// TIA Portal V20 export
// export: Created 2026-07-16T23:20:30.0572279Z, ExportSetting WithDefaults, DisplayName Totally Integrated Automation Portal, DisplayVersion V20 Update 5, DisplayName TIA Portal Openness, DisplayVersion V20 Update 4, DisplayName TIA Portal Version Control Interface, DisplayVersion V20 Update 5, DisplayName SINAMICS Startdrive Advanced, DisplayVersion V20, DisplayName SINAMICS DCC, DisplayVersion V20, DisplayName SINAMICS Startdrive G130, G150, S120, S150, SINAMICS MV, G220, S200, S210, DisplayVersion V20, DisplayName SINAMICS Startdrive G110M, G120, G120C, G120D, G120P, G115D, DisplayVersion V20, DisplayName STEP 7 Professional, DisplayVersion V20 Update 5, DisplayName STEP 7 Safety, DisplayVersion V20 Update 2, DisplayName WinCC Basic/Comfort/Advanced, DisplayVersion V20 Update 5, DisplayName WinCC Unified, DisplayVersion V20 Update 5
FUNCTION "FC_ControlMain" : Void   // FC3, LAD
TITLE = Control Main
{ S7_Optimized_Access := 'TRUE' }
VERSION : 0.1
// Control area-Main (C-109): every cross-instance fact in the project lives here (C-127) - buffer-to-instance input wiring, the sequencer/motor/pusher calls in dependency order (sequencer decides, motor and pusher obey within the same scan), inter-instance command wiring, and the buffer output map. No working logic beyond wiring, with two documented extras (C-606): the In_Cycle lamp OR (owner ruling 2026-07-16, REQ-069 - field feedbacks, not commands) and the soft-start fault-reset pass-through to DQ11 (panel provides the output; Q-14 records the open control-on question).
// stored: AutoNumber true, IsIECCheckEnabled false, SetENOAutomatically false, UDAEnableTagReadback false
BEGIN

REGION Network 1: Sequencer Input Wiring
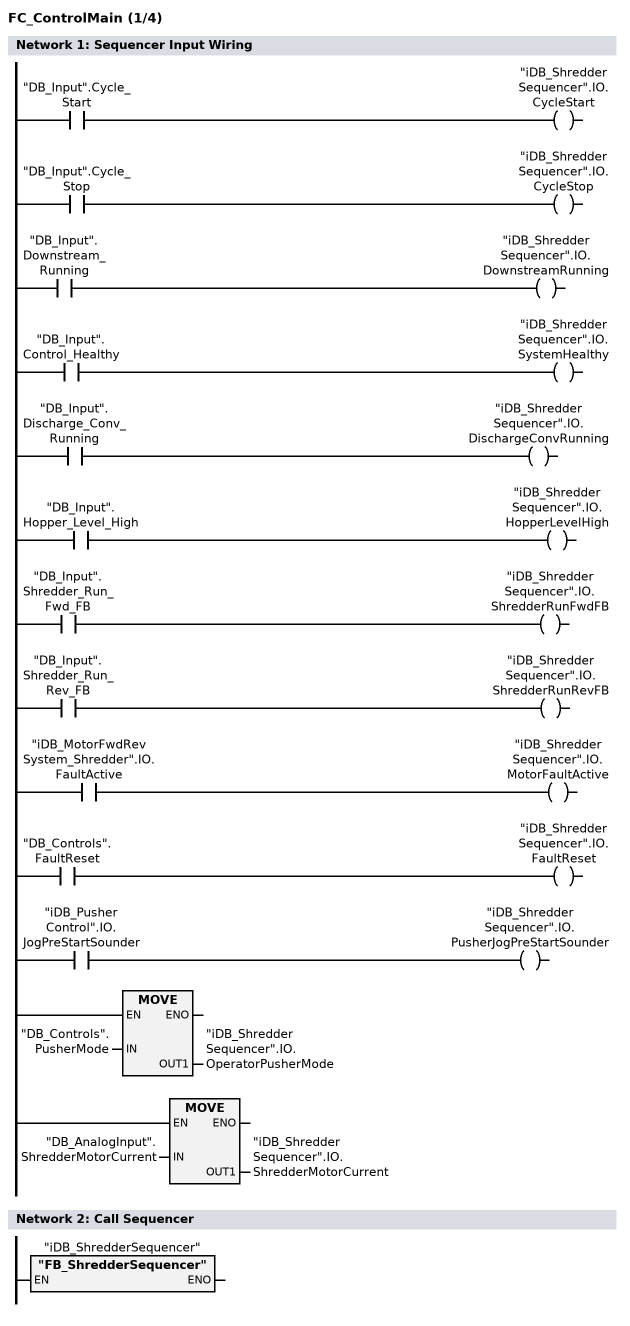
   RUNG wire#powerrail
      Contact( "DB_Input".Cycle_Start )
      Coil( "iDB_ShredderSequencer".IO.CycleStart )
   END_RUNG
   RUNG wire#powerrail
      Contact( "DB_Input".Cycle_Stop )
      Coil( "iDB_ShredderSequencer".IO.CycleStop )
   END_RUNG
   RUNG wire#powerrail
      Contact( "DB_Input".Downstream_Running )
      Coil( "iDB_ShredderSequencer".IO.DownstreamRunning )
   END_RUNG
   RUNG wire#powerrail
      Contact( "DB_Input".Control_Healthy )
      Coil( "iDB_ShredderSequencer".IO.SystemHealthy )
   END_RUNG
   RUNG wire#powerrail
      Contact( "DB_Input".Discharge_Conv_Running )
      Coil( "iDB_ShredderSequencer".IO.DischargeConvRunning )
   END_RUNG
   RUNG wire#powerrail
      Contact( "DB_Input".Hopper_Level_High )
      Coil( "iDB_ShredderSequencer".IO.HopperLevelHigh )
   END_RUNG
   RUNG wire#powerrail
      Contact( "DB_Input".Shredder_Run_Fwd_FB )
      Coil( "iDB_ShredderSequencer".IO.ShredderRunFwdFB )
   END_RUNG
   RUNG wire#powerrail
      Contact( "DB_Input".Shredder_Run_Rev_FB )
      Coil( "iDB_ShredderSequencer".IO.ShredderRunRevFB )
   END_RUNG
   RUNG wire#powerrail
      Contact( "iDB_MotorFwdRevSystem_Shredder".IO.FaultActive )
      Coil( "iDB_ShredderSequencer".IO.MotorFaultActive )
   END_RUNG
   RUNG wire#powerrail
      Contact( "DB_Controls".FaultReset )
      Coil( "iDB_ShredderSequencer".IO.FaultReset )
   END_RUNG
   RUNG wire#powerrail
      Contact( "iDB_PusherControl".IO.JogPreStartSounder )
      Coil( "iDB_ShredderSequencer".IO.PusherJogPreStartSounder )
   END_RUNG
   RUNG wire#powerrail
      Move(in := "DB_Controls".PusherMode, out1 => "iDB_ShredderSequencer".IO.OperatorPusherMode)
   END_RUNG
   RUNG wire#powerrail
      Move(in := "DB_AnalogInput".ShredderMotorCurrent, out1 => "iDB_ShredderSequencer".IO.ShredderMotorCurrent)
   END_RUNG
   // the same network as SCL:
   "iDB_ShredderSequencer".IO.CycleStart := "DB_Input".Cycle_Start;
   "iDB_ShredderSequencer".IO.CycleStop := "DB_Input".Cycle_Stop;
   "iDB_ShredderSequencer".IO.DownstreamRunning := "DB_Input".Downstream_Running;
   "iDB_ShredderSequencer".IO.SystemHealthy := "DB_Input".Control_Healthy;
   "iDB_ShredderSequencer".IO.DischargeConvRunning := "DB_Input".Discharge_Conv_Running;
   "iDB_ShredderSequencer".IO.HopperLevelHigh := "DB_Input".Hopper_Level_High;
   "iDB_ShredderSequencer".IO.ShredderRunFwdFB := "DB_Input".Shredder_Run_Fwd_FB;
   "iDB_ShredderSequencer".IO.ShredderRunRevFB := "DB_Input".Shredder_Run_Rev_FB;
   "iDB_ShredderSequencer".IO.MotorFaultActive := "iDB_MotorFwdRevSystem_Shredder".IO.FaultActive;
   "iDB_ShredderSequencer".IO.FaultReset := "DB_Controls".FaultReset;
   "iDB_ShredderSequencer".IO.PusherJogPreStartSounder := "iDB_PusherControl".IO.JogPreStartSounder;
   "iDB_ShredderSequencer".IO.OperatorPusherMode := "DB_Controls".PusherMode;
   "iDB_ShredderSequencer".IO.ShredderMotorCurrent := "DB_AnalogInput".ShredderMotorCurrent;
END_REGION

REGION Network 2: Call Sequencer
   RUNG wire#powerrail
      "iDB_ShredderSequencer"()
   END_RUNG
   // the same network as SCL:
   "iDB_ShredderSequencer"();   // "FB_ShredderSequencer"
END_REGION

REGION Network 3: MotorFwdRevSystem Wiring
   // InHand, InhibitMotor, and HandReverse are deliberate constants (C-604): unrequested imported-FB capability (hand mode, external inhibit, hand-reverse) carried disabled - design, not placeholder debt. RecentStart is armed, never driven: the sequencer's MotorStartArm (PreStart step only) ORs into the FB's own bit, and the FB's self-clear (once running or faulted - its N4 'set on start press' contract) is the only clearer, so one fresh start press arms exactly one start attempt and an E-stop or fault can never auto-restart the motor (REQ-062; replaces the RecentStart := AlwaysTrue strap that defeated the FB's semantics).
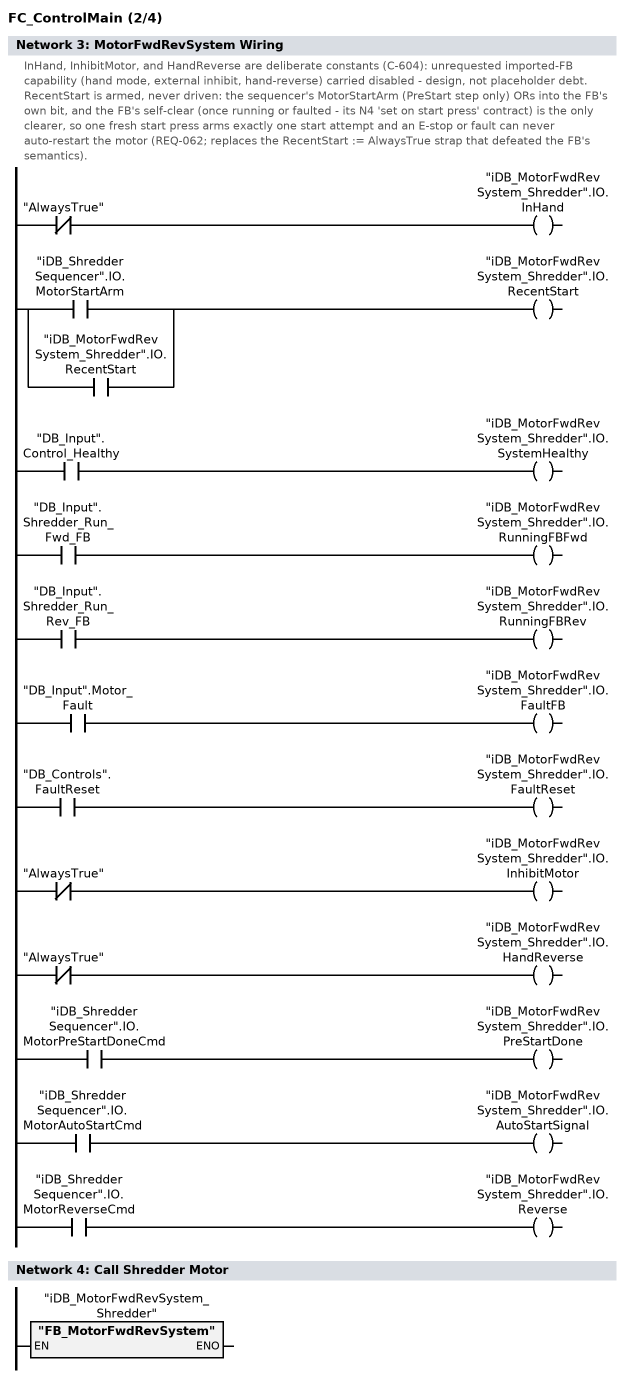
   RUNG wire#powerrail
      I_Contact( "AlwaysTrue" )
      Coil( "iDB_MotorFwdRevSystem_Shredder".IO.InHand )
   END_RUNG
   RUNG wire#powerrail
      Contact( "iDB_ShredderSequencer".IO.MotorStartArm )
      wire#w1
      Coil( "iDB_MotorFwdRevSystem_Shredder".IO.RecentStart )
   END_RUNG
   RUNG wire#powerrail
      Contact( "iDB_MotorFwdRevSystem_Shredder".IO.RecentStart )
   END_RUNG wire#w1
   RUNG wire#powerrail
      Contact( "DB_Input".Control_Healthy )
      Coil( "iDB_MotorFwdRevSystem_Shredder".IO.SystemHealthy )
   END_RUNG
   RUNG wire#powerrail
      Contact( "DB_Input".Shredder_Run_Fwd_FB )
      Coil( "iDB_MotorFwdRevSystem_Shredder".IO.RunningFBFwd )
   END_RUNG
   RUNG wire#powerrail
      Contact( "DB_Input".Shredder_Run_Rev_FB )
      Coil( "iDB_MotorFwdRevSystem_Shredder".IO.RunningFBRev )
   END_RUNG
   RUNG wire#powerrail
      Contact( "DB_Input".Motor_Fault )
      Coil( "iDB_MotorFwdRevSystem_Shredder".IO.FaultFB )
   END_RUNG
   RUNG wire#powerrail
      Contact( "DB_Controls".FaultReset )
      Coil( "iDB_MotorFwdRevSystem_Shredder".IO.FaultReset )
   END_RUNG
   RUNG wire#powerrail
      I_Contact( "AlwaysTrue" )
      Coil( "iDB_MotorFwdRevSystem_Shredder".IO.InhibitMotor )
   END_RUNG
   RUNG wire#powerrail
      I_Contact( "AlwaysTrue" )
      Coil( "iDB_MotorFwdRevSystem_Shredder".IO.HandReverse )
   END_RUNG
   RUNG wire#powerrail
      Contact( "iDB_ShredderSequencer".IO.MotorPreStartDoneCmd )
      Coil( "iDB_MotorFwdRevSystem_Shredder".IO.PreStartDone )
   END_RUNG
   RUNG wire#powerrail
      Contact( "iDB_ShredderSequencer".IO.MotorAutoStartCmd )
      Coil( "iDB_MotorFwdRevSystem_Shredder".IO.AutoStartSignal )
   END_RUNG
   RUNG wire#powerrail
      Contact( "iDB_ShredderSequencer".IO.MotorReverseCmd )
      Coil( "iDB_MotorFwdRevSystem_Shredder".IO.Reverse )
   END_RUNG
   // the same network as SCL:
   "iDB_MotorFwdRevSystem_Shredder".IO.InHand := NOT "AlwaysTrue";
   "iDB_MotorFwdRevSystem_Shredder".IO.RecentStart := "iDB_ShredderSequencer".IO.MotorStartArm OR "iDB_MotorFwdRevSystem_Shredder".IO.RecentStart;
   "iDB_MotorFwdRevSystem_Shredder".IO.SystemHealthy := "DB_Input".Control_Healthy;
   "iDB_MotorFwdRevSystem_Shredder".IO.RunningFBFwd := "DB_Input".Shredder_Run_Fwd_FB;
   "iDB_MotorFwdRevSystem_Shredder".IO.RunningFBRev := "DB_Input".Shredder_Run_Rev_FB;
   "iDB_MotorFwdRevSystem_Shredder".IO.FaultFB := "DB_Input".Motor_Fault;
   "iDB_MotorFwdRevSystem_Shredder".IO.FaultReset := "DB_Controls".FaultReset;
   "iDB_MotorFwdRevSystem_Shredder".IO.InhibitMotor := NOT "AlwaysTrue";
   "iDB_MotorFwdRevSystem_Shredder".IO.HandReverse := NOT "AlwaysTrue";
   "iDB_MotorFwdRevSystem_Shredder".IO.PreStartDone := "iDB_ShredderSequencer".IO.MotorPreStartDoneCmd;
   "iDB_MotorFwdRevSystem_Shredder".IO.AutoStartSignal := "iDB_ShredderSequencer".IO.MotorAutoStartCmd;
   "iDB_MotorFwdRevSystem_Shredder".IO.Reverse := "iDB_ShredderSequencer".IO.MotorReverseCmd;
END_REGION

REGION Network 4: Call Shredder Motor
   RUNG wire#powerrail
      "iDB_MotorFwdRevSystem_Shredder"()
   END_RUNG
   // the same network as SCL:
   "iDB_MotorFwdRevSystem_Shredder"();   // "FB_MotorFwdRevSystem"
END_REGION

REGION Network 5: PusherControl Wiring
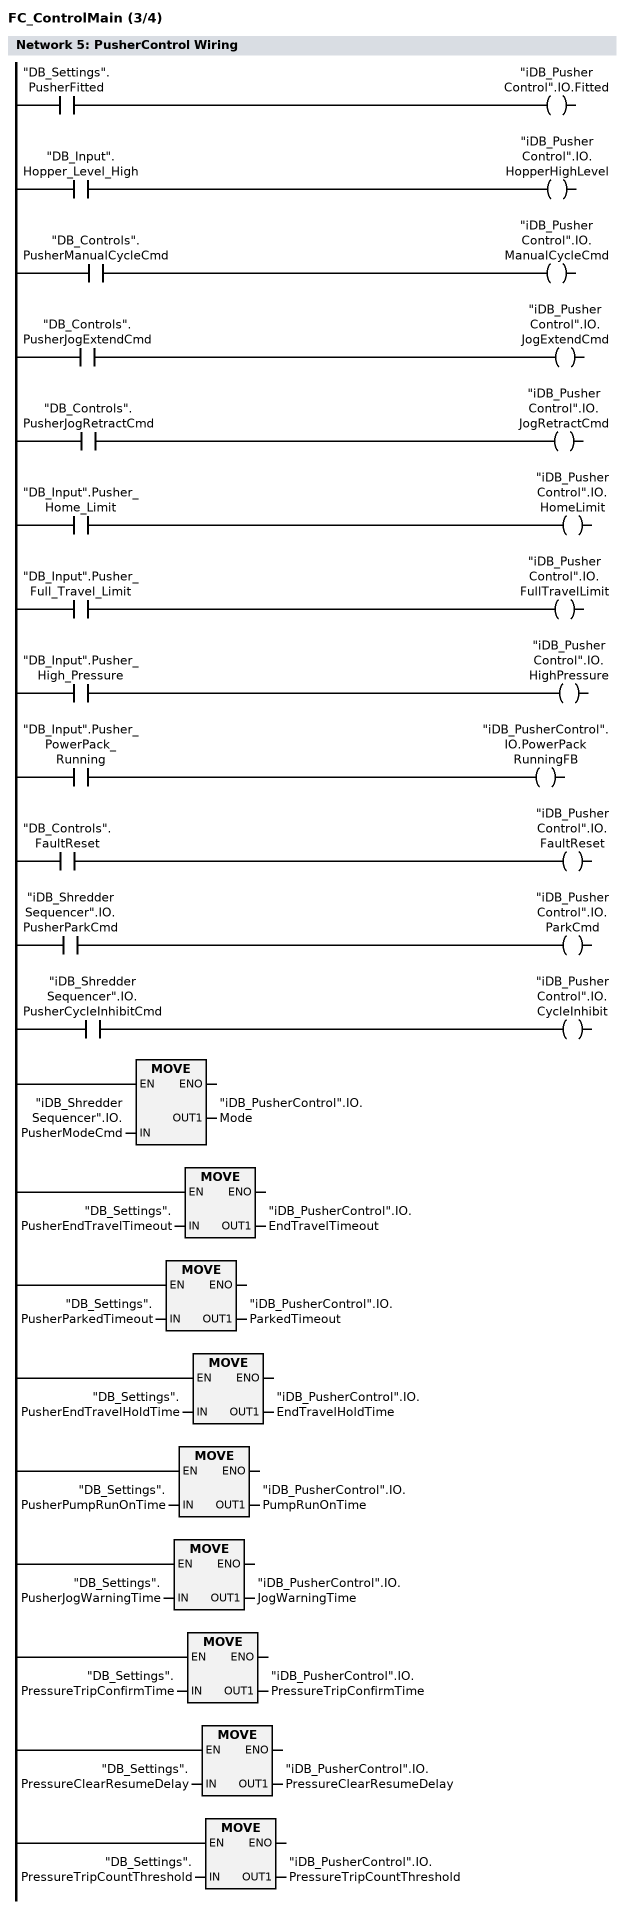
   RUNG wire#powerrail
      Contact( "DB_Settings".PusherFitted )
      Coil( "iDB_PusherControl".IO.Fitted )
   END_RUNG
   RUNG wire#powerrail
      Contact( "DB_Input".Hopper_Level_High )
      Coil( "iDB_PusherControl".IO.HopperHighLevel )
   END_RUNG
   RUNG wire#powerrail
      Contact( "DB_Controls".PusherManualCycleCmd )
      Coil( "iDB_PusherControl".IO.ManualCycleCmd )
   END_RUNG
   RUNG wire#powerrail
      Contact( "DB_Controls".PusherJogExtendCmd )
      Coil( "iDB_PusherControl".IO.JogExtendCmd )
   END_RUNG
   RUNG wire#powerrail
      Contact( "DB_Controls".PusherJogRetractCmd )
      Coil( "iDB_PusherControl".IO.JogRetractCmd )
   END_RUNG
   RUNG wire#powerrail
      Contact( "DB_Input".Pusher_Home_Limit )
      Coil( "iDB_PusherControl".IO.HomeLimit )
   END_RUNG
   RUNG wire#powerrail
      Contact( "DB_Input".Pusher_Full_Travel_Limit )
      Coil( "iDB_PusherControl".IO.FullTravelLimit )
   END_RUNG
   RUNG wire#powerrail
      Contact( "DB_Input".Pusher_High_Pressure )
      Coil( "iDB_PusherControl".IO.HighPressure )
   END_RUNG
   RUNG wire#powerrail
      Contact( "DB_Input".Pusher_PowerPack_Running )
      Coil( "iDB_PusherControl".IO.PowerPackRunningFB )
   END_RUNG
   RUNG wire#powerrail
      Contact( "DB_Controls".FaultReset )
      Coil( "iDB_PusherControl".IO.FaultReset )
   END_RUNG
   RUNG wire#powerrail
      Contact( "iDB_ShredderSequencer".IO.PusherParkCmd )
      Coil( "iDB_PusherControl".IO.ParkCmd )
   END_RUNG
   RUNG wire#powerrail
      Contact( "iDB_ShredderSequencer".IO.PusherCycleInhibitCmd )
      Coil( "iDB_PusherControl".IO.CycleInhibit )
   END_RUNG
   RUNG wire#powerrail
      Move(in := "iDB_ShredderSequencer".IO.PusherModeCmd, out1 => "iDB_PusherControl".IO.Mode)
   END_RUNG
   RUNG wire#powerrail
      Move(in := "DB_Settings".PusherEndTravelTimeout, out1 => "iDB_PusherControl".IO.EndTravelTimeout)
   END_RUNG
   RUNG wire#powerrail
      Move(in := "DB_Settings".PusherParkedTimeout, out1 => "iDB_PusherControl".IO.ParkedTimeout)
   END_RUNG
   RUNG wire#powerrail
      Move(in := "DB_Settings".PusherEndTravelHoldTime, out1 => "iDB_PusherControl".IO.EndTravelHoldTime)
   END_RUNG
   RUNG wire#powerrail
      Move(in := "DB_Settings".PusherPumpRunOnTime, out1 => "iDB_PusherControl".IO.PumpRunOnTime)
   END_RUNG
   RUNG wire#powerrail
      Move(in := "DB_Settings".PusherJogWarningTime, out1 => "iDB_PusherControl".IO.JogWarningTime)
   END_RUNG
   RUNG wire#powerrail
      Move(in := "DB_Settings".PressureTripConfirmTime, out1 => "iDB_PusherControl".IO.PressureTripConfirmTime)
   END_RUNG
   RUNG wire#powerrail
      Move(in := "DB_Settings".PressureClearResumeDelay, out1 => "iDB_PusherControl".IO.PressureClearResumeDelay)
   END_RUNG
   RUNG wire#powerrail
      Move(in := "DB_Settings".PressureTripCountThreshold, out1 => "iDB_PusherControl".IO.PressureTripCountThreshold)
   END_RUNG
   // the same network as SCL:
   "iDB_PusherControl".IO.Fitted := "DB_Settings".PusherFitted;
   "iDB_PusherControl".IO.HopperHighLevel := "DB_Input".Hopper_Level_High;
   "iDB_PusherControl".IO.ManualCycleCmd := "DB_Controls".PusherManualCycleCmd;
   "iDB_PusherControl".IO.JogExtendCmd := "DB_Controls".PusherJogExtendCmd;
   "iDB_PusherControl".IO.JogRetractCmd := "DB_Controls".PusherJogRetractCmd;
   "iDB_PusherControl".IO.HomeLimit := "DB_Input".Pusher_Home_Limit;
   "iDB_PusherControl".IO.FullTravelLimit := "DB_Input".Pusher_Full_Travel_Limit;
   "iDB_PusherControl".IO.HighPressure := "DB_Input".Pusher_High_Pressure;
   "iDB_PusherControl".IO.PowerPackRunningFB := "DB_Input".Pusher_PowerPack_Running;
   "iDB_PusherControl".IO.FaultReset := "DB_Controls".FaultReset;
   "iDB_PusherControl".IO.ParkCmd := "iDB_ShredderSequencer".IO.PusherParkCmd;
   "iDB_PusherControl".IO.CycleInhibit := "iDB_ShredderSequencer".IO.PusherCycleInhibitCmd;
   "iDB_PusherControl".IO.Mode := "iDB_ShredderSequencer".IO.PusherModeCmd;
   "iDB_PusherControl".IO.EndTravelTimeout := "DB_Settings".PusherEndTravelTimeout;
   "iDB_PusherControl".IO.ParkedTimeout := "DB_Settings".PusherParkedTimeout;
   "iDB_PusherControl".IO.EndTravelHoldTime := "DB_Settings".PusherEndTravelHoldTime;
   "iDB_PusherControl".IO.PumpRunOnTime := "DB_Settings".PusherPumpRunOnTime;
   "iDB_PusherControl".IO.JogWarningTime := "DB_Settings".PusherJogWarningTime;
   "iDB_PusherControl".IO.PressureTripConfirmTime := "DB_Settings".PressureTripConfirmTime;
   "iDB_PusherControl".IO.PressureClearResumeDelay := "DB_Settings".PressureClearResumeDelay;
   "iDB_PusherControl".IO.PressureTripCountThreshold := "DB_Settings".PressureTripCountThreshold;
END_REGION

REGION Network 6: Call Pusher
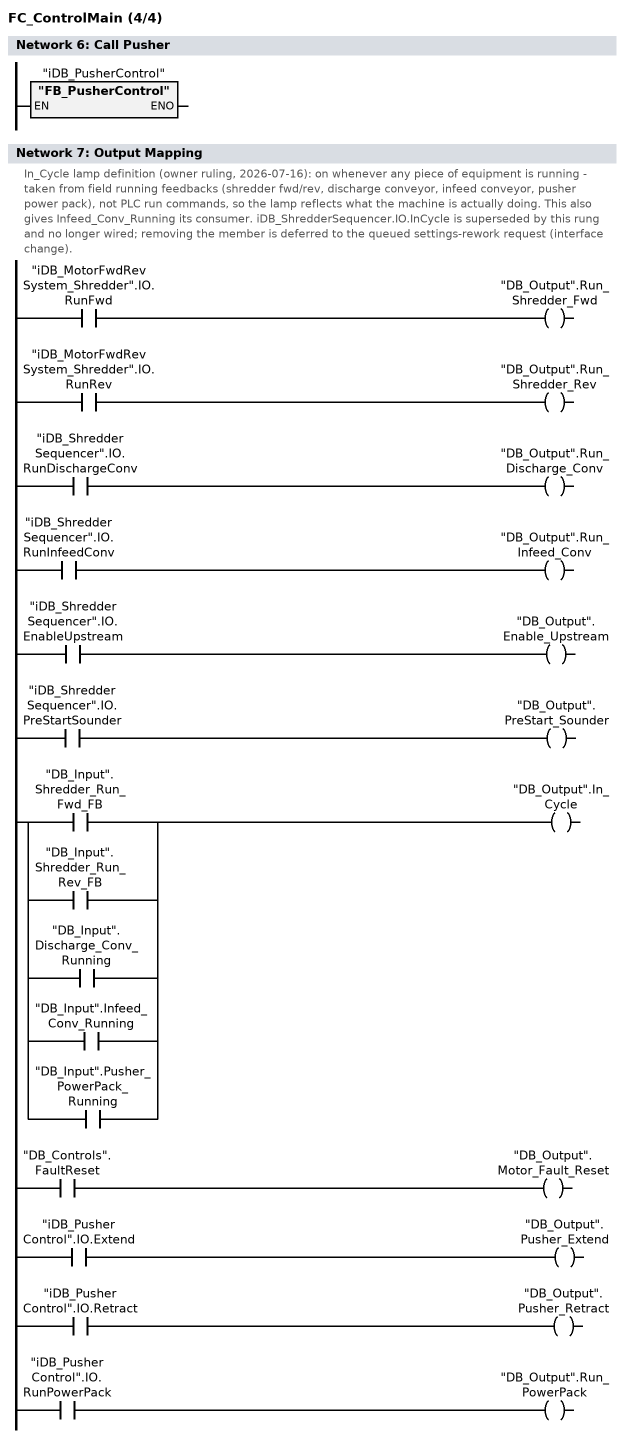
   RUNG wire#powerrail
      "iDB_PusherControl"()
   END_RUNG
   // the same network as SCL:
   "iDB_PusherControl"();   // "FB_PusherControl"
END_REGION

REGION Network 7: Output Mapping
   // In_Cycle lamp definition (owner ruling, 2026-07-16): on whenever any piece of equipment is running - taken from field running feedbacks (shredder fwd/rev, discharge conveyor, infeed conveyor, pusher power pack), not PLC run commands, so the lamp reflects what the machine is actually doing. This also gives Infeed_Conv_Running its consumer. iDB_ShredderSequencer.IO.InCycle is superseded by this rung and no longer wired; removing the member is deferred to the queued settings-rework request (interface change).
   RUNG wire#powerrail
      Contact( "iDB_MotorFwdRevSystem_Shredder".IO.RunFwd )
      Coil( "DB_Output".Run_Shredder_Fwd )
   END_RUNG
   RUNG wire#powerrail
      Contact( "iDB_MotorFwdRevSystem_Shredder".IO.RunRev )
      Coil( "DB_Output".Run_Shredder_Rev )
   END_RUNG
   RUNG wire#powerrail
      Contact( "iDB_ShredderSequencer".IO.RunDischargeConv )
      Coil( "DB_Output".Run_Discharge_Conv )
   END_RUNG
   RUNG wire#powerrail
      Contact( "iDB_ShredderSequencer".IO.RunInfeedConv )
      Coil( "DB_Output".Run_Infeed_Conv )
   END_RUNG
   RUNG wire#powerrail
      Contact( "iDB_ShredderSequencer".IO.EnableUpstream )
      Coil( "DB_Output".Enable_Upstream )
   END_RUNG
   RUNG wire#powerrail
      Contact( "iDB_ShredderSequencer".IO.PreStartSounder )
      Coil( "DB_Output".PreStart_Sounder )
   END_RUNG
   RUNG wire#powerrail
      Contact( "DB_Input".Shredder_Run_Fwd_FB )
      wire#w1
      Coil( "DB_Output".In_Cycle )
   END_RUNG
   RUNG wire#powerrail
      Contact( "DB_Input".Shredder_Run_Rev_FB )
   END_RUNG wire#w1
   RUNG wire#powerrail
      Contact( "DB_Input".Discharge_Conv_Running )
   END_RUNG wire#w1
   RUNG wire#powerrail
      Contact( "DB_Input".Infeed_Conv_Running )
   END_RUNG wire#w1
   RUNG wire#powerrail
      Contact( "DB_Input".Pusher_PowerPack_Running )
   END_RUNG wire#w1
   RUNG wire#powerrail
      Contact( "DB_Controls".FaultReset )
      Coil( "DB_Output".Motor_Fault_Reset )
   END_RUNG
   RUNG wire#powerrail
      Contact( "iDB_PusherControl".IO.Extend )
      Coil( "DB_Output".Pusher_Extend )
   END_RUNG
   RUNG wire#powerrail
      Contact( "iDB_PusherControl".IO.Retract )
      Coil( "DB_Output".Pusher_Retract )
   END_RUNG
   RUNG wire#powerrail
      Contact( "iDB_PusherControl".IO.RunPowerPack )
      Coil( "DB_Output".Run_PowerPack )
   END_RUNG
   // the same network as SCL:
   "DB_Output".Run_Shredder_Fwd := "iDB_MotorFwdRevSystem_Shredder".IO.RunFwd;
   "DB_Output".Run_Shredder_Rev := "iDB_MotorFwdRevSystem_Shredder".IO.RunRev;
   "DB_Output".Run_Discharge_Conv := "iDB_ShredderSequencer".IO.RunDischargeConv;
   "DB_Output".Run_Infeed_Conv := "iDB_ShredderSequencer".IO.RunInfeedConv;
   "DB_Output".Enable_Upstream := "iDB_ShredderSequencer".IO.EnableUpstream;
   "DB_Output".PreStart_Sounder := "iDB_ShredderSequencer".IO.PreStartSounder;
   "DB_Output".In_Cycle := "DB_Input".Shredder_Run_Fwd_FB OR "DB_Input".Shredder_Run_Rev_FB OR "DB_Input".Discharge_Conv_Running OR "DB_Input".Infeed_Conv_Running OR "DB_Input".Pusher_PowerPack_Running;
   "DB_Output".Motor_Fault_Reset := "DB_Controls".FaultReset;
   "DB_Output".Pusher_Extend := "iDB_PusherControl".IO.Extend;
   "DB_Output".Pusher_Retract := "iDB_PusherControl".IO.Retract;
   "DB_Output".Run_PowerPack := "iDB_PusherControl".IO.RunPowerPack;
END_REGION
END_FUNCTION
